Omron CX-Programmer project NewProject (CX-Programmer 9.51)

# PLC my_first_project: CP1L L
; Comment

## Program NewProgram1 (cyclic task 0)
Local symbols
button_1 0.00 BOOL  ; Comment
button_2 0.10 BOOL  ; comment
button_3 0.10 BOOL  ; comment
out_2 100.01 BOOL  ; comment
out_3 100.02 BOOL  ; comment
start W0.00 BOOL  ; comment

### Section Section1

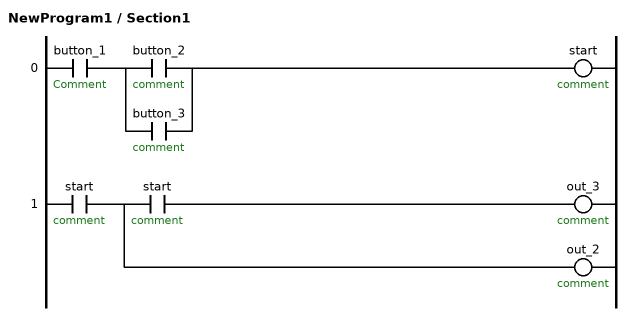
; rung 0
LD button_1  ; Comment
LD button_2  ; comment
OR button_3  ; comment
ANDLD
OUT start  ; comment
; rung 1
LD start  ; comment
OUT TR0
AND start  ; comment
OUT out_3  ; comment
LD TR0
OUT out_2  ; comment

### Section END
; rung 0
END(001)